Staubli VAL3: start.pgx

program start()
  local num l_nReturn
begin
  cls()
  userPage()
  call lib:unprotect(l_nReturn)
  put("Tool return: ")
  putln(l_nReturn)
  putln("0: no error, reboot the controller without any 'uniVAL' license in controller.cfx")
  putln("-1: VAL 3 license not enabled")
  putln("Other negative values: R&D meaning")
end
